// TIA Portal V16 export
// export: Created 2022-11-14T17:35:28.450926Z, ExportSetting WithDefaults, DisplayName Totally Integrated Automation Portal, DisplayVersion V16, DisplayName TIA Portal Version Control Interface, DisplayVersion V16, DisplayName TIA Portal Openness, DisplayVersion V16, DisplayName STEP 7 Professional, DisplayVersion V16, DisplayName STEP 7 Safety, DisplayVersion V16, DisplayName WinCC Advanced, DisplayVersion V16
FUNCTION "FC38_DisplayEsaVT505" : Void   // FC38, LAD
TITLE = Display ESA VT505 management
{ S7_Optimized_Access := 'FALSE' }
AUTHOR : Robopac
VERSION : 0.0
// stored: AutoNumber false, IsIECCheckEnabled false, SetENOAutomatically false, UDAEnableTagReadback false
   VAR_TEMP
      TempInt : Int;
   END_VAR
   VAR_TEMP   // added for the SCL form of the ladder/FBD networks
      _w1 : Bool;
      _w2 : Bool;
      _w3 : Bool;
      _w4 : Bool;
      _w5 : Bool;
   END_VAR
BEGIN

REGION Network 1: Manual(Toggle bit): Pressure plate upward/downward (Helix)
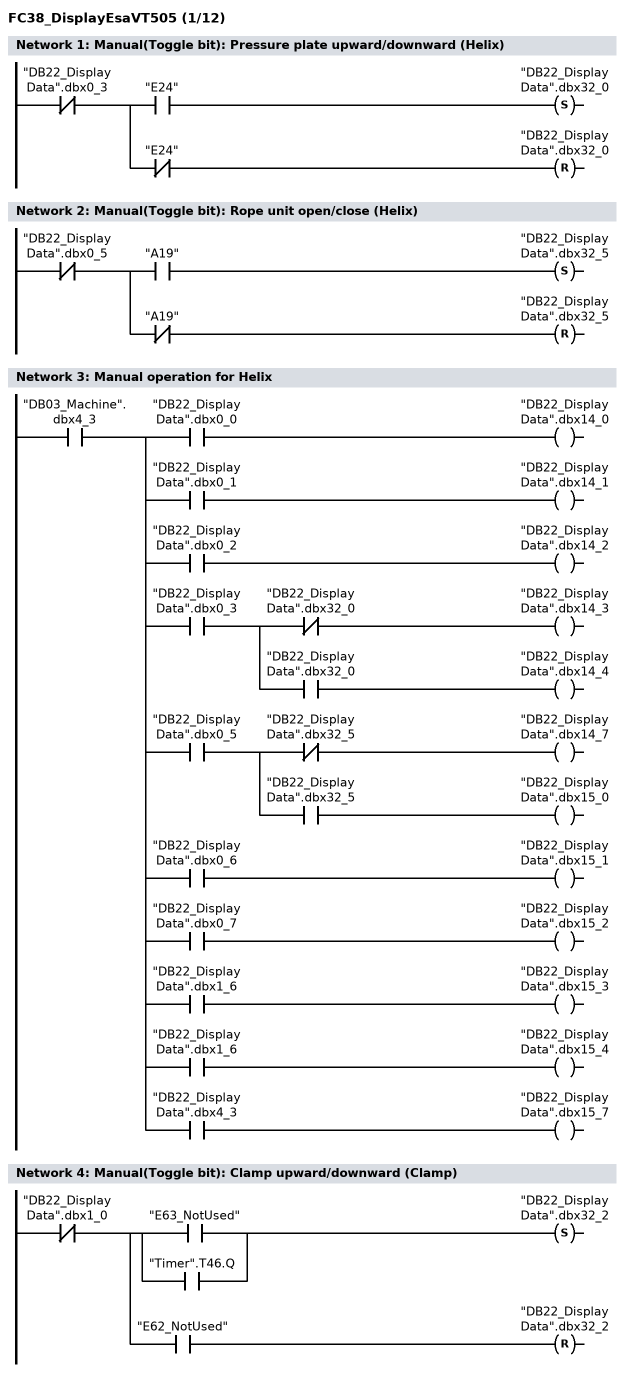
   RUNG wire#powerrail
      I_Contact( "DB22_DisplayData".dbx0_3 )
      wire#w1
      Contact( "E24" )
      S_Coil( "DB22_DisplayData".dbx32_0 )
   END_RUNG
   RUNG wire#w1
      I_Contact( "E24" )
      R_Coil( "DB22_DisplayData".dbx32_0 )
   END_RUNG
   // the same network as SCL:
   #_w1 := NOT "DB22_DisplayData".dbx0_3;
   IF #_w1 AND "E24" THEN "DB22_DisplayData".dbx32_0 := TRUE; END_IF;
   IF #_w1 AND NOT "E24" THEN "DB22_DisplayData".dbx32_0 := FALSE; END_IF;
END_REGION

REGION Network 2: Manual(Toggle bit): Rope unit open/close (Helix)
   RUNG wire#powerrail
      I_Contact( "DB22_DisplayData".dbx0_5 )
      wire#w1
      Contact( "A19" )
      S_Coil( "DB22_DisplayData".dbx32_5 )
   END_RUNG
   RUNG wire#w1
      I_Contact( "A19" )
      R_Coil( "DB22_DisplayData".dbx32_5 )
   END_RUNG
   // the same network as SCL:
   #_w1 := NOT "DB22_DisplayData".dbx0_5;
   IF #_w1 AND "A19" THEN "DB22_DisplayData".dbx32_5 := TRUE; END_IF;
   IF #_w1 AND NOT "A19" THEN "DB22_DisplayData".dbx32_5 := FALSE; END_IF;
END_REGION

REGION Network 3: Manual operation for Helix
   RUNG wire#powerrail
      Contact( "DB03_Machine".dbx4_3 )
      wire#w1
      Contact( "DB22_DisplayData".dbx0_0 )
      Coil( "DB22_DisplayData".dbx14_0 )
   END_RUNG
   RUNG wire#w1
      Contact( "DB22_DisplayData".dbx0_1 )
      Coil( "DB22_DisplayData".dbx14_1 )
   END_RUNG
   RUNG wire#w1
      Contact( "DB22_DisplayData".dbx0_2 )
      Coil( "DB22_DisplayData".dbx14_2 )
   END_RUNG
   RUNG wire#w1
      Contact( "DB22_DisplayData".dbx0_3 )
      wire#w2
      I_Contact( "DB22_DisplayData".dbx32_0 )
      Coil( "DB22_DisplayData".dbx14_3 )
   END_RUNG
   RUNG wire#w2
      Contact( "DB22_DisplayData".dbx32_0 )
      Coil( "DB22_DisplayData".dbx14_4 )
   END_RUNG
   RUNG wire#w1
      Contact( "DB22_DisplayData".dbx0_5 )
      wire#w3
      I_Contact( "DB22_DisplayData".dbx32_5 )
      Coil( "DB22_DisplayData".dbx14_7 )
   END_RUNG
   RUNG wire#w3
      Contact( "DB22_DisplayData".dbx32_5 )
      Coil( "DB22_DisplayData".dbx15_0 )
   END_RUNG
   RUNG wire#w1
      Contact( "DB22_DisplayData".dbx0_6 )
      Coil( "DB22_DisplayData".dbx15_1 )
   END_RUNG
   RUNG wire#w1
      Contact( "DB22_DisplayData".dbx0_7 )
      Coil( "DB22_DisplayData".dbx15_2 )
   END_RUNG
   RUNG wire#w1
      Contact( "DB22_DisplayData".dbx1_6 )
      Coil( "DB22_DisplayData".dbx15_3 )
   END_RUNG
   RUNG wire#w1
      Contact( "DB22_DisplayData".dbx1_6 )
      Coil( "DB22_DisplayData".dbx15_4 )
   END_RUNG
   RUNG wire#w1
      Contact( "DB22_DisplayData".dbx4_3 )
      Coil( "DB22_DisplayData".dbx15_7 )
   END_RUNG
   // the same network as SCL:
   "DB22_DisplayData".dbx14_0 := "DB03_Machine".dbx4_3 AND "DB22_DisplayData".dbx0_0;
   "DB22_DisplayData".dbx14_1 := "DB03_Machine".dbx4_3 AND "DB22_DisplayData".dbx0_1;
   "DB22_DisplayData".dbx14_2 := "DB03_Machine".dbx4_3 AND "DB22_DisplayData".dbx0_2;
   #_w1 := "DB03_Machine".dbx4_3 AND "DB22_DisplayData".dbx0_3;
   "DB22_DisplayData".dbx14_3 := #_w1 AND NOT "DB22_DisplayData".dbx32_0;
   "DB22_DisplayData".dbx14_4 := #_w1 AND "DB22_DisplayData".dbx32_0;
   #_w2 := "DB03_Machine".dbx4_3 AND "DB22_DisplayData".dbx0_5;
   "DB22_DisplayData".dbx14_7 := #_w2 AND NOT "DB22_DisplayData".dbx32_5;
   "DB22_DisplayData".dbx15_0 := #_w2 AND "DB22_DisplayData".dbx32_5;
   "DB22_DisplayData".dbx15_1 := "DB03_Machine".dbx4_3 AND "DB22_DisplayData".dbx0_6;
   "DB22_DisplayData".dbx15_2 := "DB03_Machine".dbx4_3 AND "DB22_DisplayData".dbx0_7;
   "DB22_DisplayData".dbx15_3 := "DB03_Machine".dbx4_3 AND "DB22_DisplayData".dbx1_6;
   "DB22_DisplayData".dbx15_4 := "DB03_Machine".dbx4_3 AND "DB22_DisplayData".dbx1_6;
   "DB22_DisplayData".dbx15_7 := "DB03_Machine".dbx4_3 AND "DB22_DisplayData".dbx4_3;
END_REGION

REGION Network 4: Manual(Toggle bit): Clamp upward/downward (Clamp)
   RUNG wire#powerrail
      I_Contact( "DB22_DisplayData".dbx1_0 )
      wire#w1
      Contact( "E63_NotUsed" )
      wire#w2
      S_Coil( "DB22_DisplayData".dbx32_2 )
   END_RUNG
   RUNG wire#w1
      Contact( "Timer".T46.Q )
   END_RUNG wire#w2
   RUNG wire#w1
      Contact( "E62_NotUsed" )
      R_Coil( "DB22_DisplayData".dbx32_2 )
   END_RUNG
   // the same network as SCL:
   #_w1 := NOT "DB22_DisplayData".dbx1_0;
   IF #_w1 AND ("E63_NotUsed" OR "Timer".T46.Q) THEN "DB22_DisplayData".dbx32_2 := TRUE; END_IF;
   IF #_w1 AND "E62_NotUsed" THEN "DB22_DisplayData".dbx32_2 := FALSE; END_IF;
END_REGION

REGION Network 5: Manual(Toggle bit): Welder unit upward/downward (Clamp)
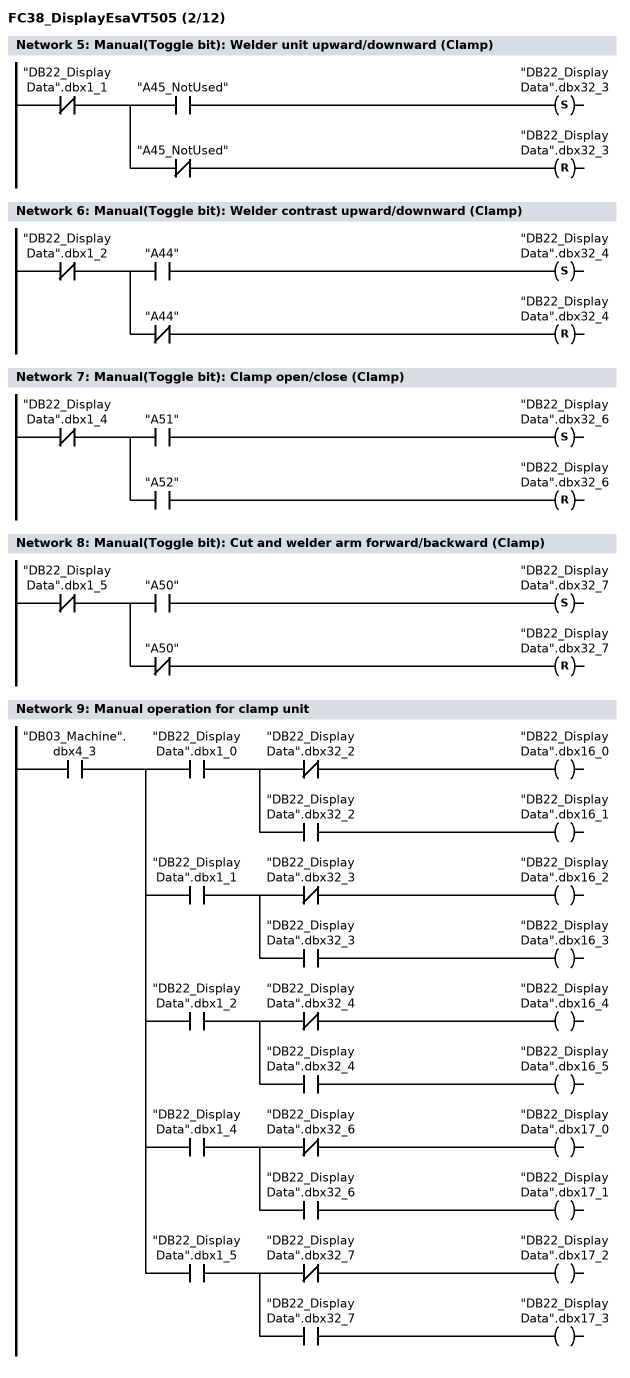
   RUNG wire#powerrail
      I_Contact( "DB22_DisplayData".dbx1_1 )
      wire#w1
      Contact( "A45_NotUsed" )
      S_Coil( "DB22_DisplayData".dbx32_3 )
   END_RUNG
   RUNG wire#w1
      I_Contact( "A45_NotUsed" )
      R_Coil( "DB22_DisplayData".dbx32_3 )
   END_RUNG
   // the same network as SCL:
   #_w1 := NOT "DB22_DisplayData".dbx1_1;
   IF #_w1 AND "A45_NotUsed" THEN "DB22_DisplayData".dbx32_3 := TRUE; END_IF;
   IF #_w1 AND NOT "A45_NotUsed" THEN "DB22_DisplayData".dbx32_3 := FALSE; END_IF;
END_REGION

REGION Network 6: Manual(Toggle bit): Welder contrast upward/downward (Clamp)
   RUNG wire#powerrail
      I_Contact( "DB22_DisplayData".dbx1_2 )
      wire#w1
      Contact( "A44" )
      S_Coil( "DB22_DisplayData".dbx32_4 )
   END_RUNG
   RUNG wire#w1
      I_Contact( "A44" )
      R_Coil( "DB22_DisplayData".dbx32_4 )
   END_RUNG
   // the same network as SCL:
   #_w1 := NOT "DB22_DisplayData".dbx1_2;
   IF #_w1 AND "A44" THEN "DB22_DisplayData".dbx32_4 := TRUE; END_IF;
   IF #_w1 AND NOT "A44" THEN "DB22_DisplayData".dbx32_4 := FALSE; END_IF;
END_REGION

REGION Network 7: Manual(Toggle bit): Clamp open/close (Clamp)
   RUNG wire#powerrail
      I_Contact( "DB22_DisplayData".dbx1_4 )
      wire#w1
      Contact( "A51" )
      S_Coil( "DB22_DisplayData".dbx32_6 )
   END_RUNG
   RUNG wire#w1
      Contact( "A52" )
      R_Coil( "DB22_DisplayData".dbx32_6 )
   END_RUNG
   // the same network as SCL:
   #_w1 := NOT "DB22_DisplayData".dbx1_4;
   IF #_w1 AND "A51" THEN "DB22_DisplayData".dbx32_6 := TRUE; END_IF;
   IF #_w1 AND "A52" THEN "DB22_DisplayData".dbx32_6 := FALSE; END_IF;
END_REGION

REGION Network 8: Manual(Toggle bit): Cut and welder arm forward/backward (Clamp)
   RUNG wire#powerrail
      I_Contact( "DB22_DisplayData".dbx1_5 )
      wire#w1
      Contact( "A50" )
      S_Coil( "DB22_DisplayData".dbx32_7 )
   END_RUNG
   RUNG wire#w1
      I_Contact( "A50" )
      R_Coil( "DB22_DisplayData".dbx32_7 )
   END_RUNG
   // the same network as SCL:
   #_w1 := NOT "DB22_DisplayData".dbx1_5;
   IF #_w1 AND "A50" THEN "DB22_DisplayData".dbx32_7 := TRUE; END_IF;
   IF #_w1 AND NOT "A50" THEN "DB22_DisplayData".dbx32_7 := FALSE; END_IF;
END_REGION

REGION Network 9: Manual operation for clamp unit
   RUNG wire#powerrail
      Contact( "DB03_Machine".dbx4_3 )
      wire#w1
      Contact( "DB22_DisplayData".dbx1_0 )
      wire#w2
      I_Contact( "DB22_DisplayData".dbx32_2 )
      Coil( "DB22_DisplayData".dbx16_0 )
   END_RUNG
   RUNG wire#w2
      Contact( "DB22_DisplayData".dbx32_2 )
      Coil( "DB22_DisplayData".dbx16_1 )
   END_RUNG
   RUNG wire#w1
      Contact( "DB22_DisplayData".dbx1_1 )
      wire#w3
      I_Contact( "DB22_DisplayData".dbx32_3 )
      Coil( "DB22_DisplayData".dbx16_2 )
   END_RUNG
   RUNG wire#w3
      Contact( "DB22_DisplayData".dbx32_3 )
      Coil( "DB22_DisplayData".dbx16_3 )
   END_RUNG
   RUNG wire#w1
      Contact( "DB22_DisplayData".dbx1_2 )
      wire#w4
      I_Contact( "DB22_DisplayData".dbx32_4 )
      Coil( "DB22_DisplayData".dbx16_4 )
   END_RUNG
   RUNG wire#w4
      Contact( "DB22_DisplayData".dbx32_4 )
      Coil( "DB22_DisplayData".dbx16_5 )
   END_RUNG
   RUNG wire#w1
      Contact( "DB22_DisplayData".dbx1_4 )
      wire#w5
      I_Contact( "DB22_DisplayData".dbx32_6 )
      Coil( "DB22_DisplayData".dbx17_0 )
   END_RUNG
   RUNG wire#w5
      Contact( "DB22_DisplayData".dbx32_6 )
      Coil( "DB22_DisplayData".dbx17_1 )
   END_RUNG
   RUNG wire#w1
      Contact( "DB22_DisplayData".dbx1_5 )
      wire#w6
      I_Contact( "DB22_DisplayData".dbx32_7 )
      Coil( "DB22_DisplayData".dbx17_2 )
   END_RUNG
   RUNG wire#w6
      Contact( "DB22_DisplayData".dbx32_7 )
      Coil( "DB22_DisplayData".dbx17_3 )
   END_RUNG
   // the same network as SCL:
   #_w1 := "DB03_Machine".dbx4_3 AND "DB22_DisplayData".dbx1_0;
   "DB22_DisplayData".dbx16_0 := #_w1 AND NOT "DB22_DisplayData".dbx32_2;
   "DB22_DisplayData".dbx16_1 := #_w1 AND "DB22_DisplayData".dbx32_2;
   #_w2 := "DB03_Machine".dbx4_3 AND "DB22_DisplayData".dbx1_1;
   "DB22_DisplayData".dbx16_2 := #_w2 AND NOT "DB22_DisplayData".dbx32_3;
   "DB22_DisplayData".dbx16_3 := #_w2 AND "DB22_DisplayData".dbx32_3;
   #_w3 := "DB03_Machine".dbx4_3 AND "DB22_DisplayData".dbx1_2;
   "DB22_DisplayData".dbx16_4 := #_w3 AND NOT "DB22_DisplayData".dbx32_4;
   "DB22_DisplayData".dbx16_5 := #_w3 AND "DB22_DisplayData".dbx32_4;
   #_w4 := "DB03_Machine".dbx4_3 AND "DB22_DisplayData".dbx1_4;
   "DB22_DisplayData".dbx17_0 := #_w4 AND NOT "DB22_DisplayData".dbx32_6;
   "DB22_DisplayData".dbx17_1 := #_w4 AND "DB22_DisplayData".dbx32_6;
   #_w5 := "DB03_Machine".dbx4_3 AND "DB22_DisplayData".dbx1_5;
   "DB22_DisplayData".dbx17_2 := #_w5 AND NOT "DB22_DisplayData".dbx32_7;
   "DB22_DisplayData".dbx17_3 := #_w5 AND "DB22_DisplayData".dbx32_7;
END_REGION

REGION Network 10: Manual(Toggle bit): Opening/closing clamp to pull top film (Top)
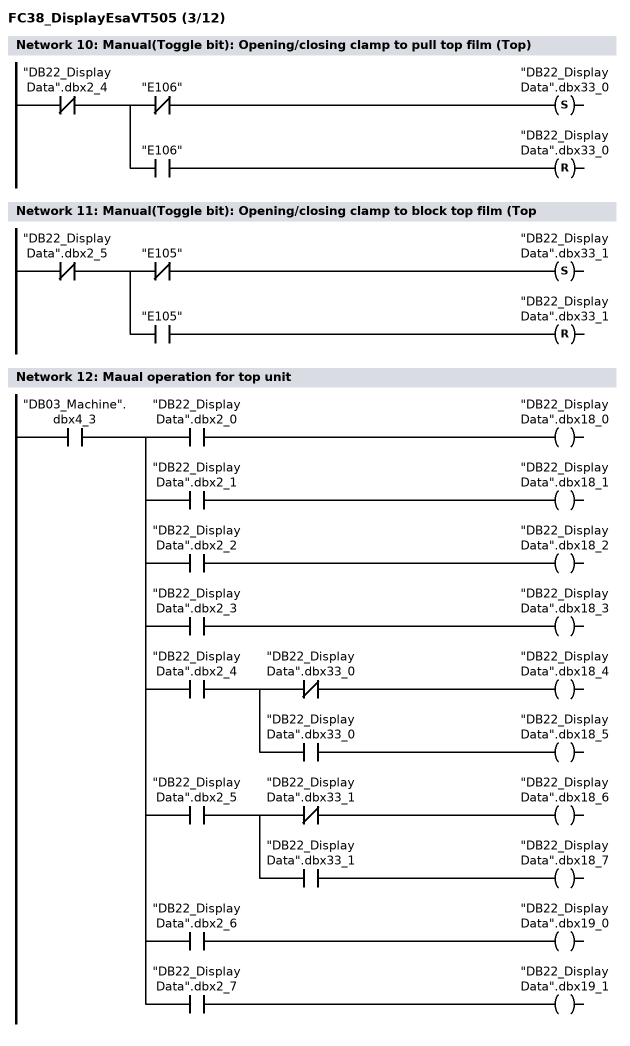
   RUNG wire#powerrail
      I_Contact( "DB22_DisplayData".dbx2_4 )
      wire#w1
      I_Contact( "E106" )
      S_Coil( "DB22_DisplayData".dbx33_0 )
   END_RUNG
   RUNG wire#w1
      Contact( "E106" )
      R_Coil( "DB22_DisplayData".dbx33_0 )
   END_RUNG
   // the same network as SCL:
   #_w1 := NOT "DB22_DisplayData".dbx2_4;
   IF #_w1 AND NOT "E106" THEN "DB22_DisplayData".dbx33_0 := TRUE; END_IF;
   IF #_w1 AND "E106" THEN "DB22_DisplayData".dbx33_0 := FALSE; END_IF;
END_REGION

REGION Network 11: Manual(Toggle bit): Opening/closing clamp to block top film (Top
   RUNG wire#powerrail
      I_Contact( "DB22_DisplayData".dbx2_5 )
      wire#w1
      I_Contact( "E105" )
      S_Coil( "DB22_DisplayData".dbx33_1 )
   END_RUNG
   RUNG wire#w1
      Contact( "E105" )
      R_Coil( "DB22_DisplayData".dbx33_1 )
   END_RUNG
   // the same network as SCL:
   #_w1 := NOT "DB22_DisplayData".dbx2_5;
   IF #_w1 AND NOT "E105" THEN "DB22_DisplayData".dbx33_1 := TRUE; END_IF;
   IF #_w1 AND "E105" THEN "DB22_DisplayData".dbx33_1 := FALSE; END_IF;
END_REGION

REGION Network 12: Maual operation for top unit
   RUNG wire#powerrail
      Contact( "DB03_Machine".dbx4_3 )
      wire#w1
      Contact( "DB22_DisplayData".dbx2_0 )
      Coil( "DB22_DisplayData".dbx18_0 )
   END_RUNG
   RUNG wire#w1
      Contact( "DB22_DisplayData".dbx2_1 )
      Coil( "DB22_DisplayData".dbx18_1 )
   END_RUNG
   RUNG wire#w1
      Contact( "DB22_DisplayData".dbx2_2 )
      Coil( "DB22_DisplayData".dbx18_2 )
   END_RUNG
   RUNG wire#w1
      Contact( "DB22_DisplayData".dbx2_3 )
      Coil( "DB22_DisplayData".dbx18_3 )
   END_RUNG
   RUNG wire#w1
      Contact( "DB22_DisplayData".dbx2_4 )
      wire#w2
      I_Contact( "DB22_DisplayData".dbx33_0 )
      Coil( "DB22_DisplayData".dbx18_4 )
   END_RUNG
   RUNG wire#w2
      Contact( "DB22_DisplayData".dbx33_0 )
      Coil( "DB22_DisplayData".dbx18_5 )
   END_RUNG
   RUNG wire#w1
      Contact( "DB22_DisplayData".dbx2_5 )
      wire#w3
      I_Contact( "DB22_DisplayData".dbx33_1 )
      Coil( "DB22_DisplayData".dbx18_6 )
   END_RUNG
   RUNG wire#w3
      Contact( "DB22_DisplayData".dbx33_1 )
      Coil( "DB22_DisplayData".dbx18_7 )
   END_RUNG
   RUNG wire#w1
      Contact( "DB22_DisplayData".dbx2_6 )
      Coil( "DB22_DisplayData".dbx19_0 )
   END_RUNG
   RUNG wire#w1
      Contact( "DB22_DisplayData".dbx2_7 )
      Coil( "DB22_DisplayData".dbx19_1 )
   END_RUNG
   // the same network as SCL:
   "DB22_DisplayData".dbx18_0 := "DB03_Machine".dbx4_3 AND "DB22_DisplayData".dbx2_0;
   "DB22_DisplayData".dbx18_1 := "DB03_Machine".dbx4_3 AND "DB22_DisplayData".dbx2_1;
   "DB22_DisplayData".dbx18_2 := "DB03_Machine".dbx4_3 AND "DB22_DisplayData".dbx2_2;
   "DB22_DisplayData".dbx18_3 := "DB03_Machine".dbx4_3 AND "DB22_DisplayData".dbx2_3;
   #_w1 := "DB03_Machine".dbx4_3 AND "DB22_DisplayData".dbx2_4;
   "DB22_DisplayData".dbx18_4 := #_w1 AND NOT "DB22_DisplayData".dbx33_0;
   "DB22_DisplayData".dbx18_5 := #_w1 AND "DB22_DisplayData".dbx33_0;
   #_w2 := "DB03_Machine".dbx4_3 AND "DB22_DisplayData".dbx2_5;
   "DB22_DisplayData".dbx18_6 := #_w2 AND NOT "DB22_DisplayData".dbx33_1;
   "DB22_DisplayData".dbx18_7 := #_w2 AND "DB22_DisplayData".dbx33_1;
   "DB22_DisplayData".dbx19_0 := "DB03_Machine".dbx4_3 AND "DB22_DisplayData".dbx2_6;
   "DB22_DisplayData".dbx19_1 := "DB03_Machine".dbx4_3 AND "DB22_DisplayData".dbx2_7;
END_REGION

REGION Network 13: Diagnostic signal conveyor
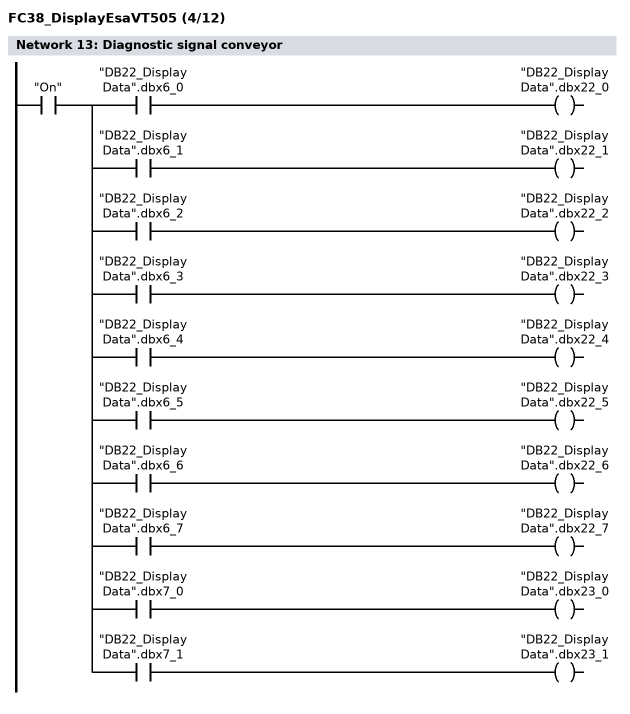
   RUNG wire#powerrail
      Contact( "On" )
      wire#w1
      Contact( "DB22_DisplayData".dbx6_0 )
      Coil( "DB22_DisplayData".dbx22_0 )
   END_RUNG
   RUNG wire#w1
      Contact( "DB22_DisplayData".dbx6_1 )
      Coil( "DB22_DisplayData".dbx22_1 )
   END_RUNG
   RUNG wire#w1
      Contact( "DB22_DisplayData".dbx6_2 )
      Coil( "DB22_DisplayData".dbx22_2 )
   END_RUNG
   RUNG wire#w1
      Contact( "DB22_DisplayData".dbx6_3 )
      Coil( "DB22_DisplayData".dbx22_3 )
   END_RUNG
   RUNG wire#w1
      Contact( "DB22_DisplayData".dbx6_4 )
      Coil( "DB22_DisplayData".dbx22_4 )
   END_RUNG
   RUNG wire#w1
      Contact( "DB22_DisplayData".dbx6_5 )
      Coil( "DB22_DisplayData".dbx22_5 )
   END_RUNG
   RUNG wire#w1
      Contact( "DB22_DisplayData".dbx6_6 )
      Coil( "DB22_DisplayData".dbx22_6 )
   END_RUNG
   RUNG wire#w1
      Contact( "DB22_DisplayData".dbx6_7 )
      Coil( "DB22_DisplayData".dbx22_7 )
   END_RUNG
   RUNG wire#w1
      Contact( "DB22_DisplayData".dbx7_0 )
      Coil( "DB22_DisplayData".dbx23_0 )
   END_RUNG
   RUNG wire#w1
      Contact( "DB22_DisplayData".dbx7_1 )
      Coil( "DB22_DisplayData".dbx23_1 )
   END_RUNG
   // the same network as SCL:
   "DB22_DisplayData".dbx22_0 := "On" AND "DB22_DisplayData".dbx6_0;
   "DB22_DisplayData".dbx22_1 := "On" AND "DB22_DisplayData".dbx6_1;
   "DB22_DisplayData".dbx22_2 := "On" AND "DB22_DisplayData".dbx6_2;
   "DB22_DisplayData".dbx22_3 := "On" AND "DB22_DisplayData".dbx6_3;
   "DB22_DisplayData".dbx22_4 := "On" AND "DB22_DisplayData".dbx6_4;
   "DB22_DisplayData".dbx22_5 := "On" AND "DB22_DisplayData".dbx6_5;
   "DB22_DisplayData".dbx22_6 := "On" AND "DB22_DisplayData".dbx6_6;
   "DB22_DisplayData".dbx22_7 := "On" AND "DB22_DisplayData".dbx6_7;
   "DB22_DisplayData".dbx23_0 := "On" AND "DB22_DisplayData".dbx7_0;
   "DB22_DisplayData".dbx23_1 := "On" AND "DB22_DisplayData".dbx7_1;
END_REGION

REGION Network 14: Diagnostic signal conveyor
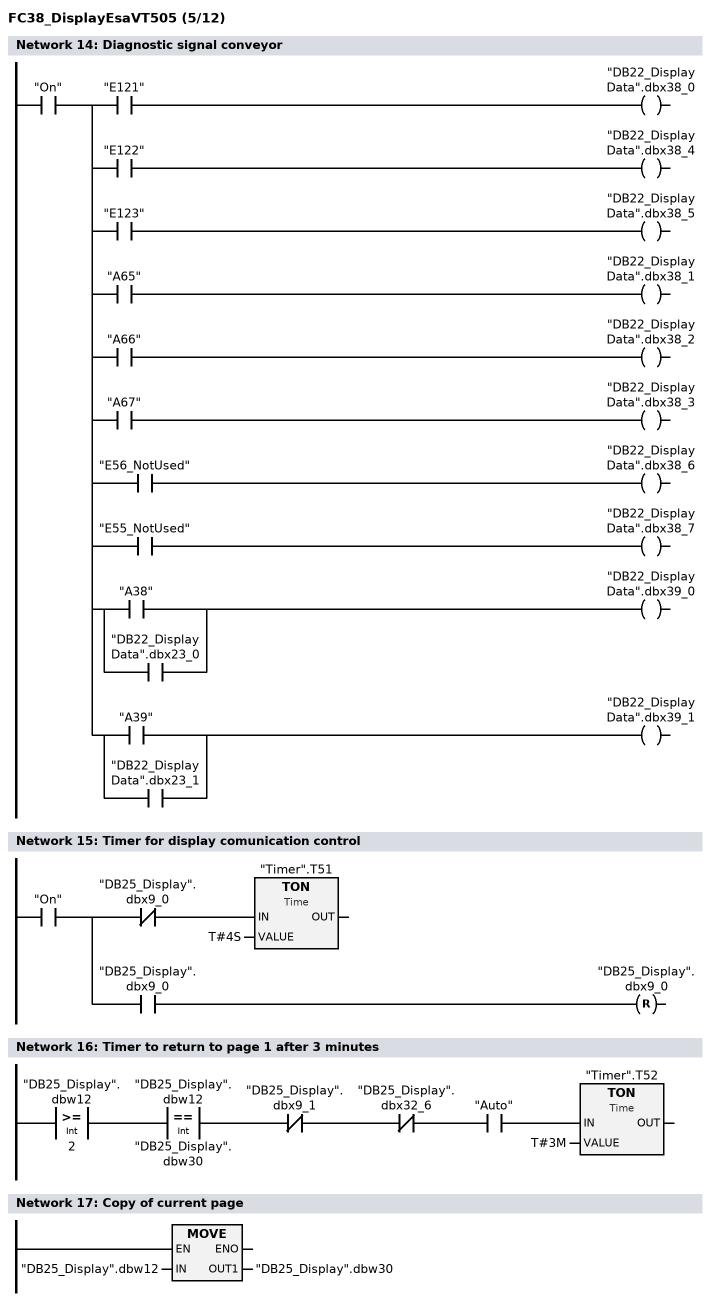
   RUNG wire#powerrail
      Contact( "On" )
      wire#w1
      Contact( "E121" )
      Coil( "DB22_DisplayData".dbx38_0 )
   END_RUNG
   RUNG wire#w1
      Contact( "E122" )
      Coil( "DB22_DisplayData".dbx38_4 )
   END_RUNG
   RUNG wire#w1
      Contact( "E123" )
      Coil( "DB22_DisplayData".dbx38_5 )
   END_RUNG
   RUNG wire#w1
      Contact( "A65" )
      Coil( "DB22_DisplayData".dbx38_1 )
   END_RUNG
   RUNG wire#w1
      Contact( "A66" )
      Coil( "DB22_DisplayData".dbx38_2 )
   END_RUNG
   RUNG wire#w1
      Contact( "A67" )
      Coil( "DB22_DisplayData".dbx38_3 )
   END_RUNG
   RUNG wire#w1
      Contact( "E56_NotUsed" )
      Coil( "DB22_DisplayData".dbx38_6 )
   END_RUNG
   RUNG wire#w1
      Contact( "E55_NotUsed" )
      Coil( "DB22_DisplayData".dbx38_7 )
   END_RUNG
   RUNG wire#w1
      Contact( "A38" )
      wire#w2
      Coil( "DB22_DisplayData".dbx39_0 )
   END_RUNG
   RUNG wire#w1
      Contact( "DB22_DisplayData".dbx23_0 )
   END_RUNG wire#w2
   RUNG wire#w1
      Contact( "A39" )
      wire#w3
      Coil( "DB22_DisplayData".dbx39_1 )
   END_RUNG
   RUNG wire#w1
      Contact( "DB22_DisplayData".dbx23_1 )
   END_RUNG wire#w3
   // the same network as SCL:
   "DB22_DisplayData".dbx38_0 := "On" AND "E121";
   "DB22_DisplayData".dbx38_4 := "On" AND "E122";
   "DB22_DisplayData".dbx38_5 := "On" AND "E123";
   "DB22_DisplayData".dbx38_1 := "On" AND "A65";
   "DB22_DisplayData".dbx38_2 := "On" AND "A66";
   "DB22_DisplayData".dbx38_3 := "On" AND "A67";
   "DB22_DisplayData".dbx38_6 := "On" AND "E56_NotUsed";
   "DB22_DisplayData".dbx38_7 := "On" AND "E55_NotUsed";
   "DB22_DisplayData".dbx39_0 := "On" AND ("A38" OR "DB22_DisplayData".dbx23_0);
   "DB22_DisplayData".dbx39_1 := "On" AND ("A39" OR "DB22_DisplayData".dbx23_1);
END_REGION

REGION Network 15: Timer for display comunication control
   "Timer".T51.TON(IN := "On" AND NOT "DB25_Display".dbx9_0, PT := T#4S);   // TON coil
   IF "On" AND "DB25_Display".dbx9_0 THEN "DB25_Display".dbx9_0 := FALSE; END_IF;
END_REGION

REGION Network 16: Timer to return to page 1 after 3 minutes
   "Timer".T52.TON(IN := ("DB25_Display".dbw12 >= 2) AND ("DB25_Display".dbw12 = "DB25_Display".dbw30) AND NOT "DB25_Display".dbx9_1 AND NOT "DB25_Display".dbx32_6 AND "Auto", PT := T#3M);   // TON coil
END_REGION

REGION Network 17: Copy of current page
   RUNG wire#powerrail
      { S7_GenerateENO := "TRUE" } Move(in := "DB25_Display".dbw12, out1 => "DB25_Display".dbw30)
   END_RUNG
   // the same network as SCL:
   "DB25_Display".dbw30 := "DB25_Display".dbw12;
END_REGION

REGION Network 18: Return to page 1 after 3 minutes
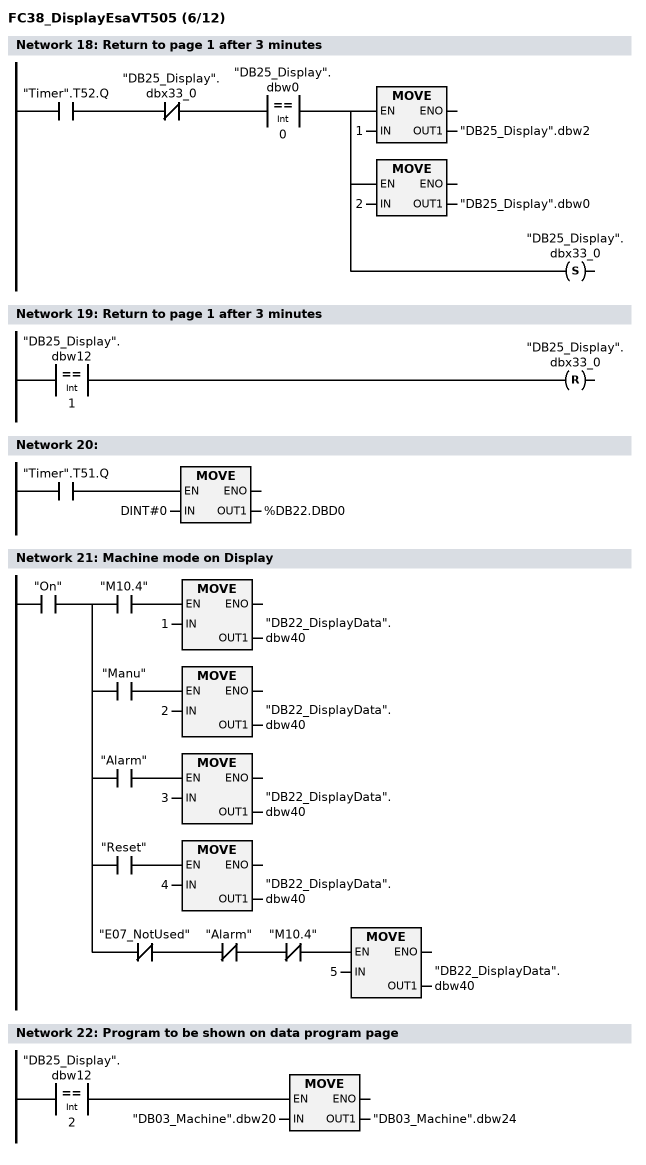
   RUNG wire#powerrail
      Contact( "Timer".T52.Q )
      I_Contact( "DB25_Display".dbx33_0 )
      { S7_Templates := "SrcType := Int" } EQ_Contact(in1 := "DB25_Display".dbw0, in2 := 0)
      wire#w1
      { S7_GenerateENO := "TRUE" } Move(in := 1, out1 => "DB25_Display".dbw2)
   END_RUNG
   RUNG wire#w1
      { S7_GenerateENO := "TRUE" } Move(in := 2, out1 => "DB25_Display".dbw0)
   END_RUNG
   RUNG wire#w1
      S_Coil( "DB25_Display".dbx33_0 )
   END_RUNG
   // the same network as SCL:
   IF "Timer".T52.Q AND NOT "DB25_Display".dbx33_0 AND ("DB25_Display".dbw0 = 0) THEN
       "DB25_Display".dbw2 := 1;
   END_IF;
   #_w1 := "Timer".T52.Q AND NOT "DB25_Display".dbx33_0 AND ("DB25_Display".dbw0 = 0);
   IF #_w1 THEN
       "DB25_Display".dbw0 := 2;
       "DB25_Display".dbx33_0 := TRUE;
   END_IF;
END_REGION

REGION Network 19: Return to page 1 after 3 minutes
   RUNG wire#powerrail
      { S7_Templates := "SrcType := Int" } EQ_Contact(in1 := "DB25_Display".dbw12, in2 := 1)
      R_Coil( "DB25_Display".dbx33_0 )
   END_RUNG
   // the same network as SCL:
   IF "DB25_Display".dbw12 = 1 THEN "DB25_Display".dbx33_0 := FALSE; END_IF;
END_REGION

REGION Network 20
   RUNG wire#powerrail
      Contact( "Timer".T51.Q )
      { S7_GenerateENO := "TRUE" } Move(in := DINT#0, out1 => %DB22.DBD0)
   END_RUNG
   // the same network as SCL:
   IF "Timer".T51.Q THEN %DB22.DBD0 := DINT#0; END_IF;
END_REGION

REGION Network 21: Machine mode on Display
   RUNG wire#powerrail
      Contact( "On" )
      wire#w1
      Contact( "M10.4" )
      { S7_GenerateENO := "TRUE" } Move(in := 1, out1 => "DB22_DisplayData".dbw40)
   END_RUNG
   RUNG wire#w1
      Contact( "Manu" )
      { S7_GenerateENO := "TRUE" } Move(in := 2, out1 => "DB22_DisplayData".dbw40)
   END_RUNG
   RUNG wire#w1
      Contact( "Alarm" )
      { S7_GenerateENO := "TRUE" } Move(in := 3, out1 => "DB22_DisplayData".dbw40)
   END_RUNG
   RUNG wire#w1
      Contact( "Reset" )
      { S7_GenerateENO := "TRUE" } Move(in := 4, out1 => "DB22_DisplayData".dbw40)
   END_RUNG
   RUNG wire#w1
      I_Contact( "E07_NotUsed" )
      I_Contact( "Alarm" )
      I_Contact( "M10.4" )
      { S7_GenerateENO := "TRUE" } Move(in := 5, out1 => "DB22_DisplayData".dbw40)
   END_RUNG
   // the same network as SCL:
   IF "On" AND "M10.4" THEN "DB22_DisplayData".dbw40 := 1; END_IF;
   IF "On" AND "Manu" THEN "DB22_DisplayData".dbw40 := 2; END_IF;
   IF "On" AND "Alarm" THEN "DB22_DisplayData".dbw40 := 3; END_IF;
   IF "On" AND "Reset" THEN "DB22_DisplayData".dbw40 := 4; END_IF;
   IF "On" AND NOT "E07_NotUsed" AND NOT "Alarm" AND NOT "M10.4" THEN "DB22_DisplayData".dbw40 := 5; END_IF;
END_REGION

REGION Network 22: Program to be shown on data program page
   RUNG wire#powerrail
      { S7_Templates := "SrcType := Int" } EQ_Contact(in1 := "DB25_Display".dbw12, in2 := 2)
      { S7_GenerateENO := "TRUE" } Move(in := "DB03_Machine".dbw20, out1 => "DB03_Machine".dbw24)
   END_RUNG
   // the same network as SCL:
   IF "DB25_Display".dbw12 = 2 THEN "DB03_Machine".dbw24 := "DB03_Machine".dbw20; END_IF;
END_REGION

REGION Network 23: Load data from data table to display area
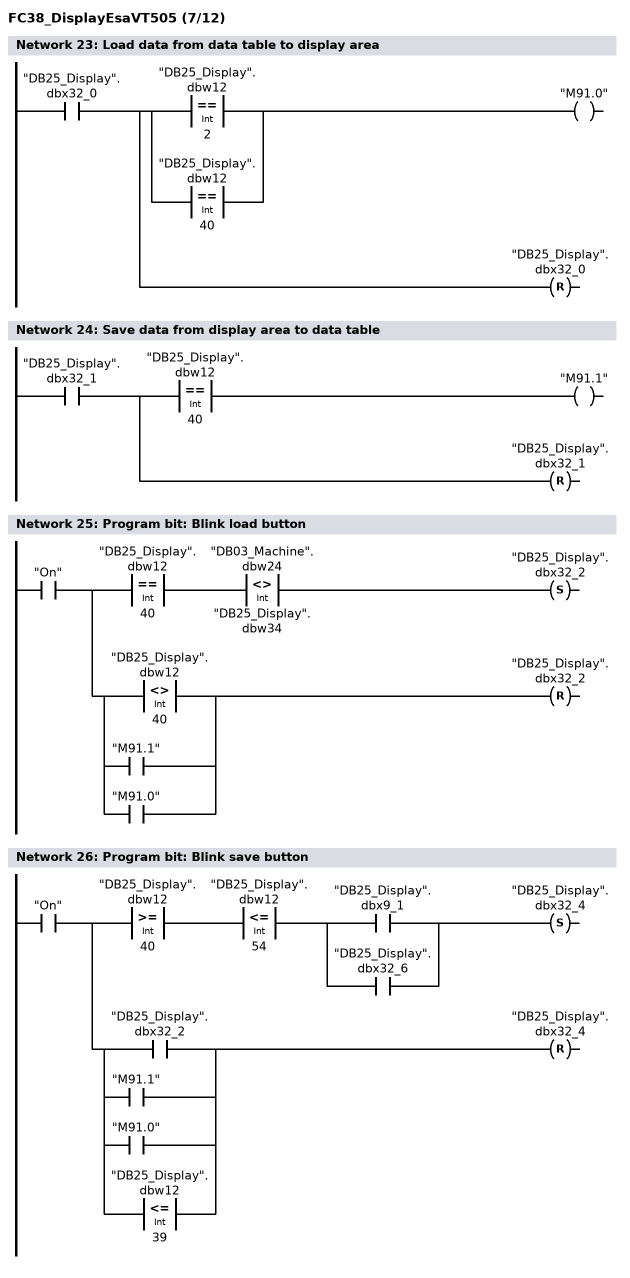
   RUNG wire#powerrail
      Contact( "DB25_Display".dbx32_0 )
      wire#w1
      { S7_Templates := "SrcType := Int" } EQ_Contact(in1 := "DB25_Display".dbw12, in2 := 2)
      wire#w2
      Coil( "M91.0" )
   END_RUNG
   RUNG wire#w1
      { S7_Templates := "SrcType := Int" } EQ_Contact(in1 := "DB25_Display".dbw12, in2 := 40)
   END_RUNG wire#w2
   RUNG wire#w1
      R_Coil( "DB25_Display".dbx32_0 )
   END_RUNG
   // the same network as SCL:
   "M91.0" := "DB25_Display".dbx32_0 AND (("DB25_Display".dbw12 = 2) OR ("DB25_Display".dbw12 = 40));
   IF "DB25_Display".dbx32_0 THEN "DB25_Display".dbx32_0 := FALSE; END_IF;
END_REGION

REGION Network 24: Save data from display area to data table
   RUNG wire#powerrail
      Contact( "DB25_Display".dbx32_1 )
      wire#w1
      { S7_Templates := "SrcType := Int" } EQ_Contact(in1 := "DB25_Display".dbw12, in2 := 40)
      Coil( "M91.1" )
   END_RUNG
   RUNG wire#w1
      R_Coil( "DB25_Display".dbx32_1 )
   END_RUNG
   // the same network as SCL:
   "M91.1" := "DB25_Display".dbx32_1 AND ("DB25_Display".dbw12 = 40);
   IF "DB25_Display".dbx32_1 THEN "DB25_Display".dbx32_1 := FALSE; END_IF;
END_REGION

REGION Network 25: Program bit: Blink load button
   RUNG wire#powerrail
      Contact( "On" )
      wire#w1
      { S7_Templates := "SrcType := Int" } EQ_Contact(in1 := "DB25_Display".dbw12, in2 := 40)
      { S7_Templates := "SrcType := Int" } NE_Contact(in1 := "DB03_Machine".dbw24, in2 := "DB25_Display".dbw34)
      S_Coil( "DB25_Display".dbx32_2 )
   END_RUNG
   RUNG wire#w1
      { S7_Templates := "SrcType := Int" } NE_Contact(in1 := "DB25_Display".dbw12, in2 := 40)
      wire#w2
      R_Coil( "DB25_Display".dbx32_2 )
   END_RUNG
   RUNG wire#w1
      Contact( "M91.1" )
   END_RUNG wire#w2
   RUNG wire#w1
      Contact( "M91.0" )
   END_RUNG wire#w2
   // the same network as SCL:
   IF "On" AND ("DB25_Display".dbw12 = 40) AND ("DB03_Machine".dbw24 <> "DB25_Display".dbw34) THEN
       "DB25_Display".dbx32_2 := TRUE;
   END_IF;
   IF "On" AND (("DB25_Display".dbw12 <> 40) OR "M91.1" OR "M91.0") THEN
       "DB25_Display".dbx32_2 := FALSE;
   END_IF;
END_REGION

REGION Network 26: Program bit: Blink save button
   RUNG wire#powerrail
      Contact( "On" )
      wire#w1
      { S7_Templates := "SrcType := Int" } GE_Contact(in1 := "DB25_Display".dbw12, in2 := 40)
      { S7_Templates := "SrcType := Int" } LE_Contact(in1 := "DB25_Display".dbw12, in2 := 54)
      wire#w2
      Contact( "DB25_Display".dbx9_1 )
      wire#w3
      S_Coil( "DB25_Display".dbx32_4 )
   END_RUNG
   RUNG wire#w2
      Contact( "DB25_Display".dbx32_6 )
   END_RUNG wire#w3
   RUNG wire#w1
      Contact( "DB25_Display".dbx32_2 )
      wire#w4
      R_Coil( "DB25_Display".dbx32_4 )
   END_RUNG
   RUNG wire#w1
      Contact( "M91.1" )
   END_RUNG wire#w4
   RUNG wire#w1
      Contact( "M91.0" )
   END_RUNG wire#w4
   RUNG wire#w1
      { S7_Templates := "SrcType := Int" } LE_Contact(in1 := "DB25_Display".dbw12, in2 := 39)
   END_RUNG wire#w4
   // the same network as SCL:
   IF "On" AND ("DB25_Display".dbw12 >= 40) AND ("DB25_Display".dbw12 <= 54) AND ("DB25_Display".dbx9_1 OR "DB25_Display".dbx32_6) THEN
       "DB25_Display".dbx32_4 := TRUE;
   END_IF;
   IF "On" AND ("DB25_Display".dbx32_2 OR "M91.1" OR "M91.0" OR ("DB25_Display".dbw12 <= 39)) THEN
       "DB25_Display".dbx32_4 := FALSE;
   END_IF;
END_REGION

REGION Network 27: Program bit:Blink load and save button
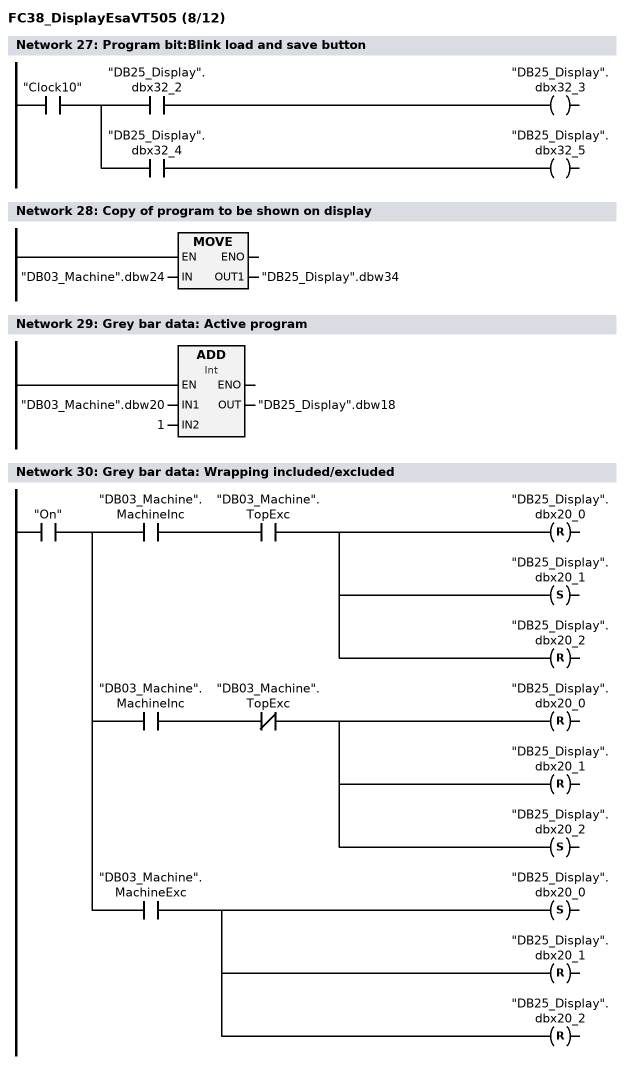
   RUNG wire#powerrail
      Contact( "Clock10" )
      wire#w1
      Contact( "DB25_Display".dbx32_2 )
      Coil( "DB25_Display".dbx32_3 )
   END_RUNG
   RUNG wire#w1
      Contact( "DB25_Display".dbx32_4 )
      Coil( "DB25_Display".dbx32_5 )
   END_RUNG
   // the same network as SCL:
   "DB25_Display".dbx32_3 := "Clock10" AND "DB25_Display".dbx32_2;
   "DB25_Display".dbx32_5 := "Clock10" AND "DB25_Display".dbx32_4;
END_REGION

REGION Network 28: Copy of program to be shown on display
   RUNG wire#powerrail
      { S7_GenerateENO := "TRUE" } Move(in := "DB03_Machine".dbw24, out1 => "DB25_Display".dbw34)
   END_RUNG
   // the same network as SCL:
   "DB25_Display".dbw34 := "DB03_Machine".dbw24;
END_REGION

REGION Network 29: Grey bar data: Active program
   RUNG wire#powerrail
      { S7_Templates := "SrcType := Int"; S7_GenerateENO := "TRUE" } Add(in1 := "DB03_Machine".dbw20, in2 := 1, out => "DB25_Display".dbw18)
   END_RUNG
   // the same network as SCL:
   "DB25_Display".dbw18 := "DB03_Machine".dbw20 + 1;
END_REGION

REGION Network 30: Grey bar data: Wrapping included/excluded
   RUNG wire#powerrail
      Contact( "On" )
      wire#w1
      Contact( "DB03_Machine".MachineInc )
      Contact( "DB03_Machine".TopExc )
      wire#w2
      R_Coil( "DB25_Display".dbx20_0 )
   END_RUNG
   RUNG wire#w2
      S_Coil( "DB25_Display".dbx20_1 )
   END_RUNG
   RUNG wire#w2
      R_Coil( "DB25_Display".dbx20_2 )
   END_RUNG
   RUNG wire#w1
      Contact( "DB03_Machine".MachineInc )
      I_Contact( "DB03_Machine".TopExc )
      wire#w3
      R_Coil( "DB25_Display".dbx20_0 )
   END_RUNG
   RUNG wire#w3
      R_Coil( "DB25_Display".dbx20_1 )
   END_RUNG
   RUNG wire#w3
      S_Coil( "DB25_Display".dbx20_2 )
   END_RUNG
   RUNG wire#w1
      Contact( "DB03_Machine".MachineExc )
      wire#w4
      S_Coil( "DB25_Display".dbx20_0 )
   END_RUNG
   RUNG wire#w4
      R_Coil( "DB25_Display".dbx20_1 )
   END_RUNG
   RUNG wire#w4
      R_Coil( "DB25_Display".dbx20_2 )
   END_RUNG
   // the same network as SCL:
   IF "On" AND "DB03_Machine".MachineInc AND "DB03_Machine".TopExc THEN
       "DB25_Display".dbx20_0 := FALSE;
       "DB25_Display".dbx20_1 := TRUE;
       "DB25_Display".dbx20_2 := FALSE;
   END_IF;
   IF "On" AND "DB03_Machine".MachineInc AND NOT "DB03_Machine".TopExc THEN
       "DB25_Display".dbx20_0 := FALSE;
       "DB25_Display".dbx20_1 := FALSE;
       "DB25_Display".dbx20_2 := TRUE;
   END_IF;
   IF "On" AND "DB03_Machine".MachineExc THEN
       "DB25_Display".dbx20_0 := TRUE;
       "DB25_Display".dbx20_1 := FALSE;
       "DB25_Display".dbx20_2 := FALSE;
   END_IF;
END_REGION

REGION Network 31: Grey bar data: Pressure plate included/excluded
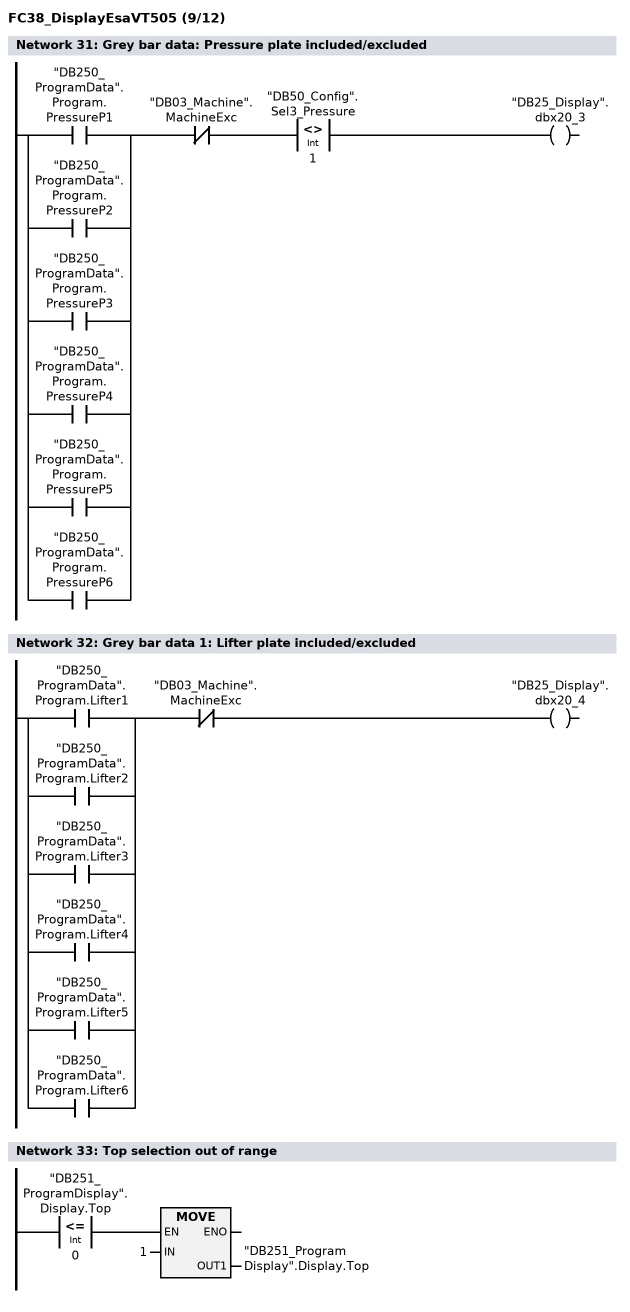
   RUNG wire#powerrail
      Contact( "DB250_ProgramData".Program.PressureP1 )
      wire#w1
      I_Contact( "DB03_Machine".MachineExc )
      { S7_Templates := "SrcType := Int" } NE_Contact(in1 := "DB50_Config".Sel3_Pressure, in2 := 1)
      Coil( "DB25_Display".dbx20_3 )
   END_RUNG
   RUNG wire#powerrail
      Contact( "DB250_ProgramData".Program.PressureP2 )
   END_RUNG wire#w1
   RUNG wire#powerrail
      Contact( "DB250_ProgramData".Program.PressureP3 )
   END_RUNG wire#w1
   RUNG wire#powerrail
      Contact( "DB250_ProgramData".Program.PressureP4 )
   END_RUNG wire#w1
   RUNG wire#powerrail
      Contact( "DB250_ProgramData".Program.PressureP5 )
   END_RUNG wire#w1
   RUNG wire#powerrail
      Contact( "DB250_ProgramData".Program.PressureP6 )
   END_RUNG wire#w1
   // the same network as SCL:
   "DB25_Display".dbx20_3 := ("DB250_ProgramData".Program.PressureP1 OR "DB250_ProgramData".Program.PressureP2 OR "DB250_ProgramData".Program.PressureP3 OR "DB250_ProgramData".Program.PressureP4 OR "DB250_ProgramData".Program.PressureP5 OR "DB250_ProgramData".Program.PressureP6) AND NOT "DB03_Machine".MachineExc AND ("DB50_Config".Sel3_Pressure <> 1);
END_REGION

REGION Network 32: Grey bar data 1: Lifter plate included/excluded
   RUNG wire#powerrail
      Contact( "DB250_ProgramData".Program.Lifter1 )
      wire#w1
      I_Contact( "DB03_Machine".MachineExc )
      Coil( "DB25_Display".dbx20_4 )
   END_RUNG
   RUNG wire#powerrail
      Contact( "DB250_ProgramData".Program.Lifter2 )
   END_RUNG wire#w1
   RUNG wire#powerrail
      Contact( "DB250_ProgramData".Program.Lifter3 )
   END_RUNG wire#w1
   RUNG wire#powerrail
      Contact( "DB250_ProgramData".Program.Lifter4 )
   END_RUNG wire#w1
   RUNG wire#powerrail
      Contact( "DB250_ProgramData".Program.Lifter5 )
   END_RUNG wire#w1
   RUNG wire#powerrail
      Contact( "DB250_ProgramData".Program.Lifter6 )
   END_RUNG wire#w1
   // the same network as SCL:
   "DB25_Display".dbx20_4 := ("DB250_ProgramData".Program.Lifter1 OR "DB250_ProgramData".Program.Lifter2 OR "DB250_ProgramData".Program.Lifter3 OR "DB250_ProgramData".Program.Lifter4 OR "DB250_ProgramData".Program.Lifter5 OR "DB250_ProgramData".Program.Lifter6) AND NOT "DB03_Machine".MachineExc;
END_REGION

REGION Network 33: Top selection out of range
   RUNG wire#powerrail
      { S7_Templates := "SrcType := Int" } LE_Contact(in1 := "DB251_ProgramDisplay".Display.Top, in2 := 0)
      { S7_GenerateENO := "TRUE" } Move(in := 1, out1 => "DB251_ProgramDisplay".Display.Top)
   END_RUNG
   // the same network as SCL:
   IF "DB251_ProgramDisplay".Display.Top <= 0 THEN "DB251_ProgramDisplay".Display.Top := 1; END_IF;
END_REGION

REGION Network 34: Top film lenght out of range
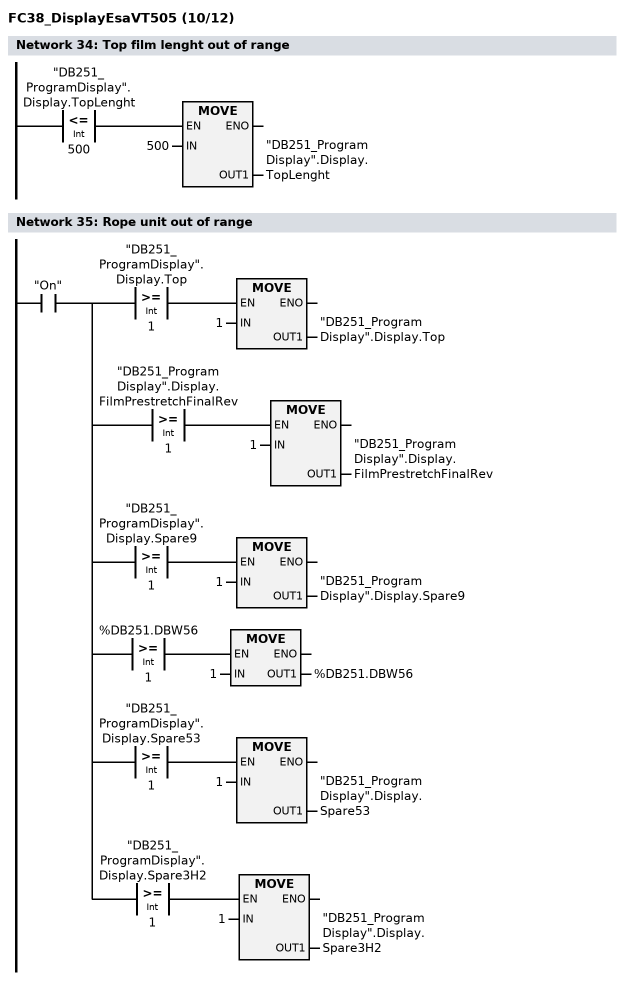
   RUNG wire#powerrail
      { S7_Templates := "SrcType := Int" } LE_Contact(in1 := "DB251_ProgramDisplay".Display.TopLenght, in2 := 500)
      { S7_GenerateENO := "TRUE" } Move(in := 500, out1 => "DB251_ProgramDisplay".Display.TopLenght)
   END_RUNG
   // the same network as SCL:
   IF "DB251_ProgramDisplay".Display.TopLenght <= 500 THEN
       "DB251_ProgramDisplay".Display.TopLenght := 500;
   END_IF;
END_REGION

REGION Network 35: Rope unit out of range
   RUNG wire#powerrail
      Contact( "On" )
      wire#w1
      { S7_Templates := "SrcType := Int" } GE_Contact(in1 := "DB251_ProgramDisplay".Display.Top, in2 := 1)
      { S7_GenerateENO := "TRUE" } Move(in := 1, out1 => "DB251_ProgramDisplay".Display.Top)
   END_RUNG
   RUNG wire#w1
      { S7_Templates := "SrcType := Int" } GE_Contact(in1 := "DB251_ProgramDisplay".Display.FilmPrestretchFinalRev, in2 := 1)
      { S7_GenerateENO := "TRUE" } Move(in := 1, out1 => "DB251_ProgramDisplay".Display.FilmPrestretchFinalRev)
   END_RUNG
   RUNG wire#w1
      { S7_Templates := "SrcType := Int" } GE_Contact(in1 := "DB251_ProgramDisplay".Display.Spare9, in2 := 1)
      { S7_GenerateENO := "TRUE" } Move(in := 1, out1 => "DB251_ProgramDisplay".Display.Spare9)
   END_RUNG
   RUNG wire#w1
      { S7_Templates := "SrcType := Int" } GE_Contact(in1 := %DB251.DBW56, in2 := 1)
      { S7_GenerateENO := "TRUE" } Move(in := 1, out1 => %DB251.DBW56)
   END_RUNG
   RUNG wire#w1
      { S7_Templates := "SrcType := Int" } GE_Contact(in1 := "DB251_ProgramDisplay".Display.Spare53, in2 := 1)
      { S7_GenerateENO := "TRUE" } Move(in := 1, out1 => "DB251_ProgramDisplay".Display.Spare53)
   END_RUNG
   RUNG wire#w1
      { S7_Templates := "SrcType := Int" } GE_Contact(in1 := "DB251_ProgramDisplay".Display.Spare3H2, in2 := 1)
      { S7_GenerateENO := "TRUE" } Move(in := 1, out1 => "DB251_ProgramDisplay".Display.Spare3H2)
   END_RUNG
   // the same network as SCL:
   IF "On" AND ("DB251_ProgramDisplay".Display.Top >= 1) THEN
       "DB251_ProgramDisplay".Display.Top := 1;
   END_IF;
   IF "On" AND ("DB251_ProgramDisplay".Display.FilmPrestretchFinalRev >= 1) THEN
       "DB251_ProgramDisplay".Display.FilmPrestretchFinalRev := 1;
   END_IF;
   IF "On" AND ("DB251_ProgramDisplay".Display.Spare9 >= 1) THEN
       "DB251_ProgramDisplay".Display.Spare9 := 1;
   END_IF;
   IF "On" AND (%DB251.DBW56 >= 1) THEN %DB251.DBW56 := 1; END_IF;
   IF "On" AND ("DB251_ProgramDisplay".Display.Spare53 >= 1) THEN
       "DB251_ProgramDisplay".Display.Spare53 := 1;
   END_IF;
   IF "On" AND ("DB251_ProgramDisplay".Display.Spare3H2 >= 1) THEN
       "DB251_ProgramDisplay".Display.Spare3H2 := 1;
   END_IF;
END_REGION

REGION Network 36: Rope unit out of range
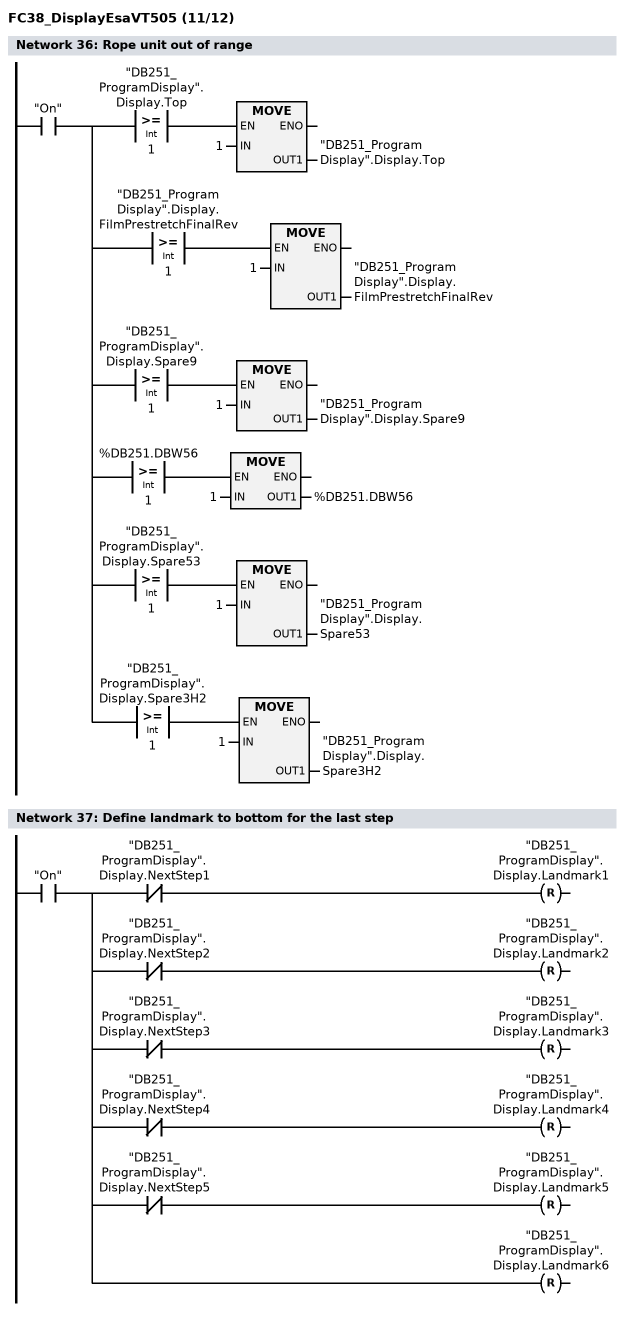
   RUNG wire#powerrail
      Contact( "On" )
      wire#w1
      { S7_Templates := "SrcType := Int" } GE_Contact(in1 := "DB251_ProgramDisplay".Display.Top, in2 := 1)
      { S7_GenerateENO := "TRUE" } Move(in := 1, out1 => "DB251_ProgramDisplay".Display.Top)
   END_RUNG
   RUNG wire#w1
      { S7_Templates := "SrcType := Int" } GE_Contact(in1 := "DB251_ProgramDisplay".Display.FilmPrestretchFinalRev, in2 := 1)
      { S7_GenerateENO := "TRUE" } Move(in := 1, out1 => "DB251_ProgramDisplay".Display.FilmPrestretchFinalRev)
   END_RUNG
   RUNG wire#w1
      { S7_Templates := "SrcType := Int" } GE_Contact(in1 := "DB251_ProgramDisplay".Display.Spare9, in2 := 1)
      { S7_GenerateENO := "TRUE" } Move(in := 1, out1 => "DB251_ProgramDisplay".Display.Spare9)
   END_RUNG
   RUNG wire#w1
      { S7_Templates := "SrcType := Int" } GE_Contact(in1 := %DB251.DBW56, in2 := 1)
      { S7_GenerateENO := "TRUE" } Move(in := 1, out1 => %DB251.DBW56)
   END_RUNG
   RUNG wire#w1
      { S7_Templates := "SrcType := Int" } GE_Contact(in1 := "DB251_ProgramDisplay".Display.Spare53, in2 := 1)
      { S7_GenerateENO := "TRUE" } Move(in := 1, out1 => "DB251_ProgramDisplay".Display.Spare53)
   END_RUNG
   RUNG wire#w1
      { S7_Templates := "SrcType := Int" } GE_Contact(in1 := "DB251_ProgramDisplay".Display.Spare3H2, in2 := 1)
      { S7_GenerateENO := "TRUE" } Move(in := 1, out1 => "DB251_ProgramDisplay".Display.Spare3H2)
   END_RUNG
   // the same network as SCL:
   IF "On" AND ("DB251_ProgramDisplay".Display.Top >= 1) THEN
       "DB251_ProgramDisplay".Display.Top := 1;
   END_IF;
   IF "On" AND ("DB251_ProgramDisplay".Display.FilmPrestretchFinalRev >= 1) THEN
       "DB251_ProgramDisplay".Display.FilmPrestretchFinalRev := 1;
   END_IF;
   IF "On" AND ("DB251_ProgramDisplay".Display.Spare9 >= 1) THEN
       "DB251_ProgramDisplay".Display.Spare9 := 1;
   END_IF;
   IF "On" AND (%DB251.DBW56 >= 1) THEN %DB251.DBW56 := 1; END_IF;
   IF "On" AND ("DB251_ProgramDisplay".Display.Spare53 >= 1) THEN
       "DB251_ProgramDisplay".Display.Spare53 := 1;
   END_IF;
   IF "On" AND ("DB251_ProgramDisplay".Display.Spare3H2 >= 1) THEN
       "DB251_ProgramDisplay".Display.Spare3H2 := 1;
   END_IF;
END_REGION

REGION Network 37: Define landmark to bottom for the last step
   RUNG wire#powerrail
      Contact( "On" )
      wire#w1
      I_Contact( "DB251_ProgramDisplay".Display.NextStep1 )
      R_Coil( "DB251_ProgramDisplay".Display.Landmark1 )
   END_RUNG
   RUNG wire#w1
      I_Contact( "DB251_ProgramDisplay".Display.NextStep2 )
      R_Coil( "DB251_ProgramDisplay".Display.Landmark2 )
   END_RUNG
   RUNG wire#w1
      I_Contact( "DB251_ProgramDisplay".Display.NextStep3 )
      R_Coil( "DB251_ProgramDisplay".Display.Landmark3 )
   END_RUNG
   RUNG wire#w1
      I_Contact( "DB251_ProgramDisplay".Display.NextStep4 )
      R_Coil( "DB251_ProgramDisplay".Display.Landmark4 )
   END_RUNG
   RUNG wire#w1
      I_Contact( "DB251_ProgramDisplay".Display.NextStep5 )
      R_Coil( "DB251_ProgramDisplay".Display.Landmark5 )
   END_RUNG
   RUNG wire#w1
      R_Coil( "DB251_ProgramDisplay".Display.Landmark6 )
   END_RUNG
   // the same network as SCL:
   IF "On" AND NOT "DB251_ProgramDisplay".Display.NextStep1 THEN
       "DB251_ProgramDisplay".Display.Landmark1 := FALSE;
   END_IF;
   IF "On" AND NOT "DB251_ProgramDisplay".Display.NextStep2 THEN
       "DB251_ProgramDisplay".Display.Landmark2 := FALSE;
   END_IF;
   IF "On" AND NOT "DB251_ProgramDisplay".Display.NextStep3 THEN
       "DB251_ProgramDisplay".Display.Landmark3 := FALSE;
   END_IF;
   IF "On" AND NOT "DB251_ProgramDisplay".Display.NextStep4 THEN
       "DB251_ProgramDisplay".Display.Landmark4 := FALSE;
   END_IF;
   IF "On" AND NOT "DB251_ProgramDisplay".Display.NextStep5 THEN
       "DB251_ProgramDisplay".Display.Landmark5 := FALSE;
   END_IF;
   IF "On" THEN "DB251_ProgramDisplay".Display.Landmark6 := FALSE; END_IF;
END_REGION

REGION Network 38
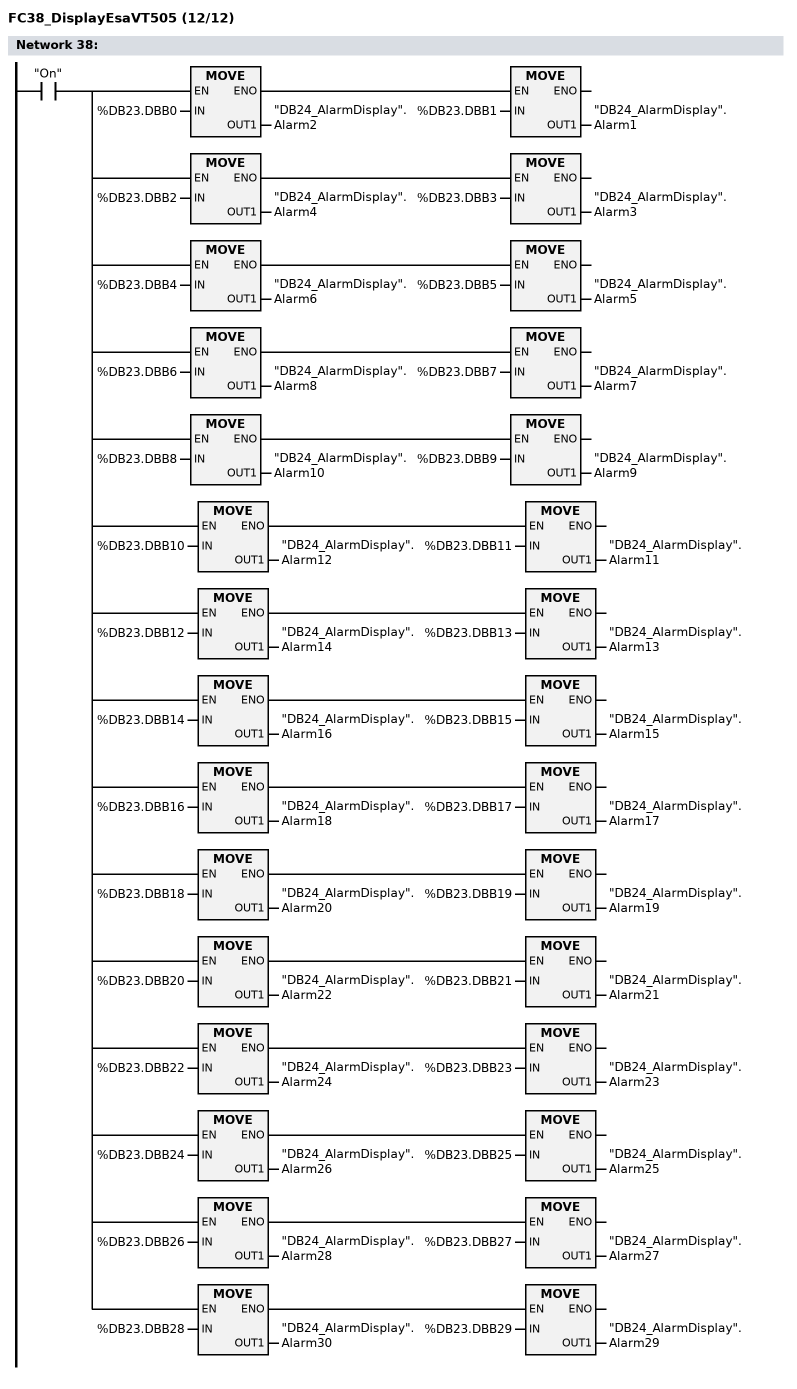
   RUNG wire#powerrail
      Contact( "On" )
      wire#w1
      { S7_GenerateENO := "TRUE" } Move(in := %DB23.DBB0, out1 => "DB24_AlarmDisplay".Alarm2)
      { S7_GenerateENO := "TRUE" } Move(in := %DB23.DBB1, out1 => "DB24_AlarmDisplay".Alarm1)
   END_RUNG
   RUNG wire#w1
      { S7_GenerateENO := "TRUE" } Move(in := %DB23.DBB2, out1 => "DB24_AlarmDisplay".Alarm4)
      { S7_GenerateENO := "TRUE" } Move(in := %DB23.DBB3, out1 => "DB24_AlarmDisplay".Alarm3)
   END_RUNG
   RUNG wire#w1
      { S7_GenerateENO := "TRUE" } Move(in := %DB23.DBB4, out1 => "DB24_AlarmDisplay".Alarm6)
      { S7_GenerateENO := "TRUE" } Move(in := %DB23.DBB5, out1 => "DB24_AlarmDisplay".Alarm5)
   END_RUNG
   RUNG wire#w1
      { S7_GenerateENO := "TRUE" } Move(in := %DB23.DBB6, out1 => "DB24_AlarmDisplay".Alarm8)
      { S7_GenerateENO := "TRUE" } Move(in := %DB23.DBB7, out1 => "DB24_AlarmDisplay".Alarm7)
   END_RUNG
   RUNG wire#w1
      { S7_GenerateENO := "TRUE" } Move(in := %DB23.DBB8, out1 => "DB24_AlarmDisplay".Alarm10)
      { S7_GenerateENO := "TRUE" } Move(in := %DB23.DBB9, out1 => "DB24_AlarmDisplay".Alarm9)
   END_RUNG
   RUNG wire#w1
      { S7_GenerateENO := "TRUE" } Move(in := %DB23.DBB10, out1 => "DB24_AlarmDisplay".Alarm12)
      { S7_GenerateENO := "TRUE" } Move(in := %DB23.DBB11, out1 => "DB24_AlarmDisplay".Alarm11)
   END_RUNG
   RUNG wire#w1
      { S7_GenerateENO := "TRUE" } Move(in := %DB23.DBB12, out1 => "DB24_AlarmDisplay".Alarm14)
      { S7_GenerateENO := "TRUE" } Move(in := %DB23.DBB13, out1 => "DB24_AlarmDisplay".Alarm13)
   END_RUNG
   RUNG wire#w1
      { S7_GenerateENO := "TRUE" } Move(in := %DB23.DBB14, out1 => "DB24_AlarmDisplay".Alarm16)
      { S7_GenerateENO := "TRUE" } Move(in := %DB23.DBB15, out1 => "DB24_AlarmDisplay".Alarm15)
   END_RUNG
   RUNG wire#w1
      { S7_GenerateENO := "TRUE" } Move(in := %DB23.DBB16, out1 => "DB24_AlarmDisplay".Alarm18)
      { S7_GenerateENO := "TRUE" } Move(in := %DB23.DBB17, out1 => "DB24_AlarmDisplay".Alarm17)
   END_RUNG
   RUNG wire#w1
      { S7_GenerateENO := "TRUE" } Move(in := %DB23.DBB18, out1 => "DB24_AlarmDisplay".Alarm20)
      { S7_GenerateENO := "TRUE" } Move(in := %DB23.DBB19, out1 => "DB24_AlarmDisplay".Alarm19)
   END_RUNG
   RUNG wire#w1
      { S7_GenerateENO := "TRUE" } Move(in := %DB23.DBB20, out1 => "DB24_AlarmDisplay".Alarm22)
      { S7_GenerateENO := "TRUE" } Move(in := %DB23.DBB21, out1 => "DB24_AlarmDisplay".Alarm21)
   END_RUNG
   RUNG wire#w1
      { S7_GenerateENO := "TRUE" } Move(in := %DB23.DBB22, out1 => "DB24_AlarmDisplay".Alarm24)
      { S7_GenerateENO := "TRUE" } Move(in := %DB23.DBB23, out1 => "DB24_AlarmDisplay".Alarm23)
   END_RUNG
   RUNG wire#w1
      { S7_GenerateENO := "TRUE" } Move(in := %DB23.DBB24, out1 => "DB24_AlarmDisplay".Alarm26)
      { S7_GenerateENO := "TRUE" } Move(in := %DB23.DBB25, out1 => "DB24_AlarmDisplay".Alarm25)
   END_RUNG
   RUNG wire#w1
      { S7_GenerateENO := "TRUE" } Move(in := %DB23.DBB26, out1 => "DB24_AlarmDisplay".Alarm28)
      { S7_GenerateENO := "TRUE" } Move(in := %DB23.DBB27, out1 => "DB24_AlarmDisplay".Alarm27)
   END_RUNG
   RUNG wire#w1
      { S7_GenerateENO := "TRUE" } Move(in := %DB23.DBB28, out1 => "DB24_AlarmDisplay".Alarm30)
      { S7_GenerateENO := "TRUE" } Move(in := %DB23.DBB29, out1 => "DB24_AlarmDisplay".Alarm29)
   END_RUNG
   // the same network as SCL:
   // ENO of a box is taken as its EN; it also drops when the box reports an error
   IF "On" THEN
       "DB24_AlarmDisplay".Alarm2 := %DB23.DBB0;
       "DB24_AlarmDisplay".Alarm1 := %DB23.DBB1;
       "DB24_AlarmDisplay".Alarm4 := %DB23.DBB2;
       "DB24_AlarmDisplay".Alarm3 := %DB23.DBB3;
       "DB24_AlarmDisplay".Alarm6 := %DB23.DBB4;
       "DB24_AlarmDisplay".Alarm5 := %DB23.DBB5;
       "DB24_AlarmDisplay".Alarm8 := %DB23.DBB6;
       "DB24_AlarmDisplay".Alarm7 := %DB23.DBB7;
       "DB24_AlarmDisplay".Alarm10 := %DB23.DBB8;
       "DB24_AlarmDisplay".Alarm9 := %DB23.DBB9;
       "DB24_AlarmDisplay".Alarm12 := %DB23.DBB10;
       "DB24_AlarmDisplay".Alarm11 := %DB23.DBB11;
       "DB24_AlarmDisplay".Alarm14 := %DB23.DBB12;
       "DB24_AlarmDisplay".Alarm13 := %DB23.DBB13;
       "DB24_AlarmDisplay".Alarm16 := %DB23.DBB14;
       "DB24_AlarmDisplay".Alarm15 := %DB23.DBB15;
       "DB24_AlarmDisplay".Alarm18 := %DB23.DBB16;
       "DB24_AlarmDisplay".Alarm17 := %DB23.DBB17;
       "DB24_AlarmDisplay".Alarm20 := %DB23.DBB18;
       "DB24_AlarmDisplay".Alarm19 := %DB23.DBB19;
       "DB24_AlarmDisplay".Alarm22 := %DB23.DBB20;
       "DB24_AlarmDisplay".Alarm21 := %DB23.DBB21;
       "DB24_AlarmDisplay".Alarm24 := %DB23.DBB22;
       "DB24_AlarmDisplay".Alarm23 := %DB23.DBB23;
       "DB24_AlarmDisplay".Alarm26 := %DB23.DBB24;
       "DB24_AlarmDisplay".Alarm25 := %DB23.DBB25;
       "DB24_AlarmDisplay".Alarm28 := %DB23.DBB26;
       "DB24_AlarmDisplay".Alarm27 := %DB23.DBB27;
       "DB24_AlarmDisplay".Alarm30 := %DB23.DBB28;
       "DB24_AlarmDisplay".Alarm29 := %DB23.DBB29;
   END_IF;
END_REGION
END_FUNCTION
